TYPE ST_CtrlInLoadstacker :
STRUCT
	DeleteAssignmentData			: BOOL := TRUE;		//overwrite Assignment ID with UNKNOWN when zone being occupied.
	DestinationFunction			: E_FunctionNumber := E_FunctionNumber.F_BEGIN_FUNCTION;
	DestinationZone				: INT :=1;
	TU_Type						: INT :=0;			
	Mode						: E_LSPM_Mode; 	// Which (E_LSPM_Mode) mode should the pallet magazine run in (Destack/Stack/SendPallet/SendStack)
END_STRUCT
END_TYPE

(* stored: Version 1.1.0.1, ProductVersion 3.1.4024.9
   DUT ST_CtrlInLoadstacker: Id {107fcfa1-7f3d-45ec-b0cd-c31bf252e9fc} *)
